// TwinCAT 3 PLC project Untitled1
// ProgramVersion: 3.1.4020.10
// libraries:
//   Tc2_Standard, * (Beckhoff Automation GmbH)
//   Tc2_System, * (Beckhoff Automation GmbH)
//   Tc3_Module, * (Beckhoff Automation GmbH)
//   VisuDialogs, * (System)
// project tree:
//   / GlobalTextList.TcGTLO, PlcTask.TcTTO, Visualization Manager.TcVMO (not stored)
//   POUs/ FB_PIZZA_OVEN.TcPOU, MAIN.TcPOU
//   VISUs/ Visualization_1.TcVIS
// real-time tasks:
//   TASK PlcTask: cycle T#10ms, priority 20, ADS port 350

CONFIGURATION Untitled1
    RESOURCE PLC ON TwinCAT3
        TASK PlcTask(INTERVAL := T#10ms, PRIORITY := 20);
        PROGRAM MAIN WITH PlcTask : MAIN;
    END_RESOURCE
END_CONFIGURATION

// ---- POUs/MAIN.TcPOU
PROGRAM MAIN
VAR

	fbMyPizzaOven : FB_PIZZA_OVEN;

	fbMyPizzaOven1 : FB_PIZZA_OVEN;
	
	bLoadPizza   : BOOL;
	bRemovePizza : BOOL;	
	
END_VAR



fbMyPizzaOven(bLoadPizza:= bLoadPizza, bRemovePizza:=bRemovePizza);


fbMyPizzaOven1(bLoadPizza:= bLoadPizza, bRemovePizza:=bRemovePizza);

END_PROGRAM

// ---- POUs/FB_PIZZA_OVEN.TcPOU
FUNCTION_BLOCK FB_PIZZA_OVEN
VAR_INPUT

	
	bLoadPizza   : BOOL;
	bRemovePizza : BOOL;

	

	

END_VAR
VAR_OUTPUT

	iTotalPizzasCooked	: UDINT;
	bBuzzer 	 : BOOL;
	bLight		 : BOOL;
END_VAR
VAR
	
	fbLoad_RTRIG : R_TRIG;
	fbRemove_RTRIG : R_TRIG;

	bPizzaInOven : BOOL;
	bPizzaOnDeck : BOOL;
	bPizzaDone	 : BOOL;
	
	
	iState		: DINT;
	sStateDesc	: STRING;	
	
	fbMyTimer	 : TON;


END_VAR


fbLoad_RTRIG(clk := bLoadPizza);
IF fbLoad_RTRIG.Q THEN
	bPizzaOnDeck := TRUE;
END_IF

fbRemove_RTRIG(clk := bRemovePizza);
IF fbRemove_RTRIG.Q THEN
	bPizzaDone := FALSE;
END_IF

IF bPizzaOnDeck AND NOT bPizzaInOven THEN
	bPizzaOnDeck := FALSE;
	bPizzaInOven := TRUE;
END_IF

CASE iState OF
	
// wait for pizza in Oven
	0: 
		sStateDesc := 'Waiting on Pizza now';
		IF bPizzaInOven THEN
			iState := 10;
		END_IF
	
// we got a pizza in the oven!		
	10: 
		sStateDesc := 'Baking that Pizza now';
		fbMyTimer(IN:=TRUE,PT := T#3S);
		IF fbMyTimer.Q THEN
			fbMyTimer(IN:=FALSE);
			iState := 20;
		END_IF
	
// can we move the pizza out of the oven?
	20:
		sStateDesc := 'Pizza is done!';
		IF NOT bPizzaDone THEN 
			bPizzaDone := TRUE;
			bPizzaInOven := FALSE;
			bBuzzer := FALSE;
			iState := 30;
		ELSE 
			bBuzzer := TRUE;
			
		END_IF
	
	30:
		sStateDesc := 'Invalid State';
		iTotalPizzasCooked := iTotalPizzasCooked + 1;
		iState := 0;
	ELSE;
		
END_CASE

END_FUNCTION_BLOCK

// ---- GlobalTextList.TcGTLO
TEXTLIST GlobalTextList
  5 = '%d'
  3 = 'Buzzer'
  2 = 'Elapsed Time: %s'
  0 = 'Insert Pizza'
  7 = 'Load Pizza'
  4 = 'MAIN.iTotalPizzasCooked'
  8 = 'Package Pizza'
  1 = 'Remove Pizza'
  6 = 'Status: %s'
END_TEXTLIST

// ---- VISUs/Visualization_1.TcVIS
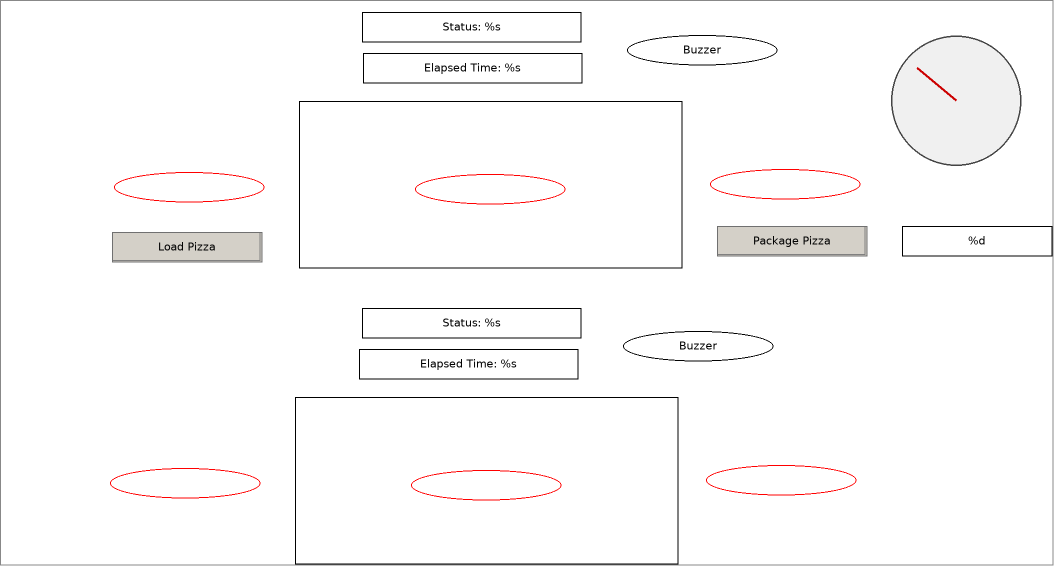
VISUALIZATION Visualization_1  // 1054x566
    Rectangle (299,101 383x167)
    Button (112,232 150x30), "Load Pizza"
        tap MAIN.bLoadPizza
        OnMouseDown: execute {  }
    Button (717,226 150x30), "Package Pizza"
        tap MAIN.bRemovePizza
        OnMouseDown: execute {  }
    Ellipse (415,174 150x30), colour toggle: MAIN.fbMyPizzaOven1.bBuzzer, invisible if: NOT MAIN.fbMyPizzaOven1.bPizzaInOven
    Rectangle (363,53 219x30), "Elapsed Time: %s", text variable: MAIN.fbMyPizzaOven1.fbMyTimer.ET
    Ellipse (627,35 150x30), "Buzzer", colour toggle: MAIN.fbMyPizzaOven1.bBuzzer
    Meter360 (891,26 130x149), value: MAIN.fbMyPizzaOven1.iTotalPizzasCooked, style: Meter-Meter360-Gray, scale format: %.1f, scale 0..20
    Rectangle (902,226 150x30), "%d", text variable: MAIN.fbMyPizzaOven1.iTotalPizzasCooked
    Rectangle (362,12 219x30), "Status: %s", text variable: MAIN.fbMyPizzaOven1.sStateDesc
    Ellipse (114,172 150x30), invisible if: NOT MAIN.fbMyPizzaOven1.bPizzaOnDeck
    Ellipse (710,169 150x30), invisible if: NOT MAIN.fbMyPizzaOven1.bPizzaDone
    Rectangle (295,397 383x167)
    Ellipse (411,470 150x30), colour toggle: MAIN.fbMyPizzaOven1.bBuzzer, invisible if: NOT MAIN.fbMyPizzaOven1.bPizzaInOven
    Rectangle (359,349 219x30), "Elapsed Time: %s", text variable: MAIN.fbMyPizzaOven1.fbMyTimer.ET
    Ellipse (623,331 150x30), "Buzzer", colour toggle: MAIN.fbMyPizzaOven1.bBuzzer
    Rectangle (362,308 219x30), "Status: %s", text variable: MAIN.fbMyPizzaOven1.sStateDesc
    Ellipse (110,468 150x30), invisible if: NOT MAIN.fbMyPizzaOven1.bPizzaOnDeck
    Ellipse (706,465 150x30), invisible if: NOT MAIN.fbMyPizzaOven1.bPizzaDone
END_VISUALIZATION
